// TIA Portal V20 export
DATA_BLOCK "SBK02"   // DB323
// stored: MemoryReserve 100
   VAR
      "SCS BOX SCS MODE SLELECT SS.SETUP" : Bool := FALSE;
      "SCS BOX SCS MODE SLELECT SS.DISABLE" : Bool := FALSE;
      "EMO05 CH.A" : Bool := FALSE;
      SPARE : Bool := FALSE;
      "SCS BOX SCS MODE SLELECT SS.AUTO" : Bool := TRUE;
      SPARE_1 : Bool := FALSE;
      "EMO05 CH.B" : Bool := FALSE;
      SPARE_2 : Bool := FALSE;
      "SCS BOX SCS MODE SELECT PL.PENDANT" : Bool := FALSE;
      "SCS BOX SCS MODE SELECT PL.DISABLE" : Bool := FALSE;
      SPARE_3 : Bool;
   END_VAR
BEGIN
END_DATA_BLOCK
